// TIA Portal V20 export
DATA_BLOCK "SP504"   // DB340
// stored: MemoryReserve 100
   VAR
      SPARE : Bool := FALSE;
      SPARE_1 : Bool := FALSE;
      "ANODE ALIGN VISION CONTROLLER TRIGEER IN" : Bool := FALSE;
      "STACK VISION CONTROLLER TRIGEER IN" : Bool := FALSE;
      "CATHODE ALIGN VISION CONTROLLER TRIGEER IN" : Bool := FALSE;
      SPARE_2 : Bool := FALSE;
   END_VAR
BEGIN
END_DATA_BLOCK
